// SIMATIC STEP 7 (V5.x) project Estacion completa
// CPU: CPU 314IFM
// station: P_ADR_BUS
// station: Hardware
// station: Equipo SIMATIC 300
// program: Programa S7(2)

// (several symbol tables fit these blocks; global names not applied)

DATA_BLOCK DB 1
VERSION : 0.1
  STRUCT
   M10 : BOOL ;	//Variable comodín provisional
  END_STRUCT ;	
BEGIN
END_DATA_BLOCK

ORGANIZATION_BLOCK OB 1
TITLE = "Main Program Sweep (Cycle)"
VERSION : 0.1
VAR_TEMP
  OB1_EV_CLASS : BYTE ;	//Bits 0-3 = 1 (Coming event), Bits 4-7 = 1 (Event class 1)
  OB1_SCAN_1 : BYTE ;	//1 (Cold restart scan 1 of OB 1), 3 (Scan 2-n of OB 1)
  OB1_PRIORITY : BYTE ;	//Priority of OB Execution
  OB1_OB_NUMBR : BYTE ;	//1 (Organization block 1, OB1)
  OB1_RESERVED_1 : BYTE ;	//Reserved for system
  OB1_RESERVED_2 : BYTE ;	//Reserved for system
  OB1_PREV_CYCLE : INT ;	//Cycle time of previous OB1 scan (milliseconds)
  OB1_MIN_CYCLE : INT ;	//Minimum cycle time of OB1 (milliseconds)
  OB1_MAX_CYCLE : INT ;	//Maximum cycle time of OB1 (milliseconds)
  OB1_DATE_TIME : DATE_AND_TIME ;	//Date and time OB1 started
END_VAR
BEGIN
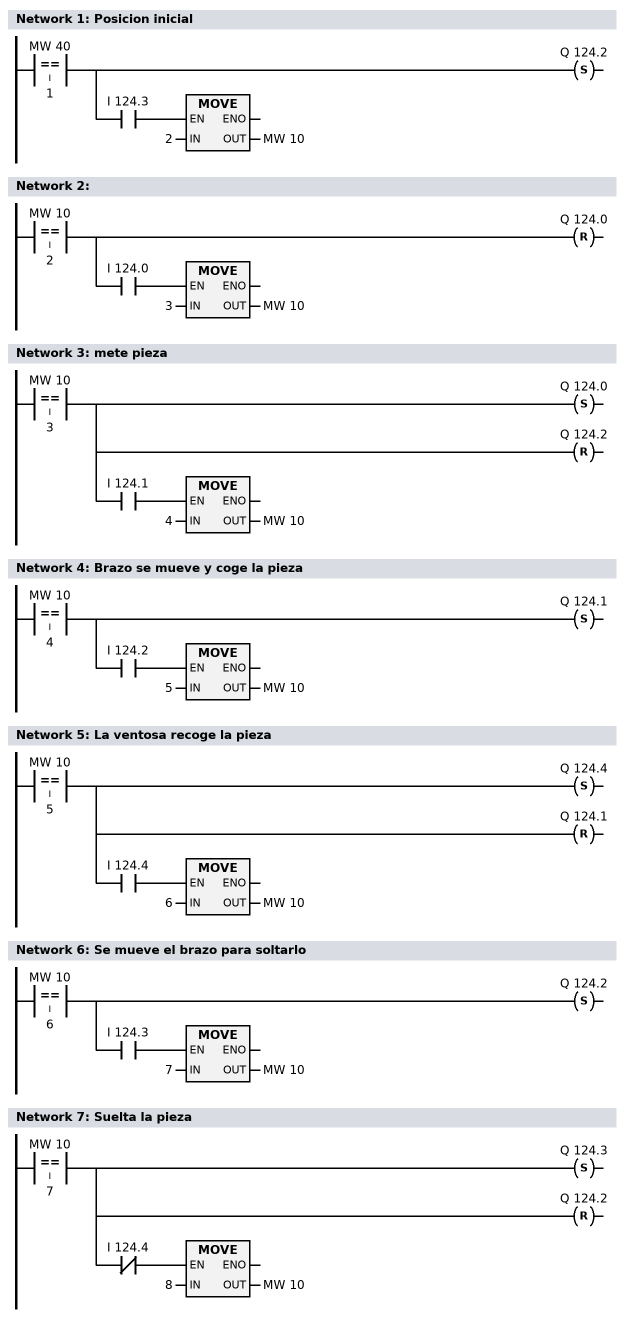
NETWORK
TITLE = Posicion inicial
      L     MW 40;
      L     1;
      ==I;
      =     L 20.0;
      A     L 20.0;
      BLD   102;
      S     Q 124.2;
      A     L 20.0;
      A     I 124.3;
      JNB   _001;
      L     2;
      T     MW 10;
_001: NOP   0;
NETWORK
TITLE =
      L     MW 10;
      L     2;
      ==I;
      =     L 20.0;
      A     L 20.0;
      BLD   102;
      R     Q 124.0;
      A     L 20.0;
      A     I 124.0;
      JNB   _002;
      L     3;
      T     MW 10;
_002: NOP   0;
NETWORK
TITLE = mete pieza
      L     MW 10;
      L     3;
      ==I;
      =     L 20.0;
      A     L 20.0;
      BLD   102;
      S     Q 124.0;
      A     L 20.0;
      BLD   102;
      R     Q 124.2;
      A     L 20.0;
      A     I 124.1;
      JNB   _003;
      L     4;
      T     MW 10;
_003: NOP   0;
NETWORK
TITLE = Brazo se mueve y coge la pieza
      L     MW 10;
      L     4;
      ==I;
      =     L 20.0;
      A     L 20.0;
      BLD   102;
      S     Q 124.1;
      A     L 20.0;
      A     I 124.2;
      JNB   _004;
      L     5;
      T     MW 10;
_004: NOP   0;
NETWORK
TITLE = La ventosa recoge la pieza
      L     MW 10;
      L     5;
      ==I;
      =     L 20.0;
      A     L 20.0;
      BLD   102;
      S     Q 124.4;
      A     L 20.0;
      BLD   102;
      R     Q 124.1;
      A     L 20.0;
      A     I 124.4;
      JNB   _005;
      L     6;
      T     MW 10;
_005: NOP   0;
NETWORK
TITLE = Se mueve el brazo para soltarlo
      L     MW 10;
      L     6;
      ==I;
      =     L 20.0;
      A     L 20.0;
      BLD   102;
      S     Q 124.2;
      A     L 20.0;
      A     I 124.3;
      JNB   _006;
      L     7;
      T     MW 10;
_006: NOP   0;
NETWORK
TITLE = Suelta la pieza
      L     MW 10;
      L     7;
      ==I;
      =     L 20.0;
      A     L 20.0;
      BLD   102;
      S     Q 124.3;
      A     L 20.0;
      BLD   102;
      R     Q 124.2;
      A     L 20.0;
      AN    I 124.4;
      JNB   _007;
      L     8;
      T     MW 10;
_007: NOP   0;
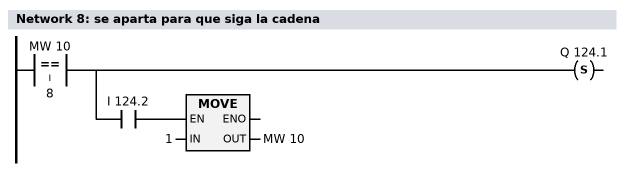
NETWORK
TITLE = se aparta para que siga la cadena
      L     MW 10;
      L     8;
      ==I;
      =     L 20.0;
      A     L 20.0;
      BLD   102;
      S     Q 124.1;
      A     L 20.0;
      A     I 124.2;
      JNB   _008;
      L     1;
      T     MW 10;
_008: NOP   0;
NETWORK
TITLE =
NETWORK
TITLE =
NETWORK
TITLE =
NETWORK
TITLE =
END_ORGANIZATION_BLOCK

SYMBOL_TABLE
"ATT"	FC 84	FC 84	// Add to Table
"CYCL_EXC"	OB 1	OB 1	// Cycle Execution
"COMPLETE RESTART"	OB 100	OB 100	// Complete Restart
"VAT_1"	VAT 1	
END_SYMBOL_TABLE

FUNCTION_BLOCK FB 1
VERSION : 0.1
BEGIN
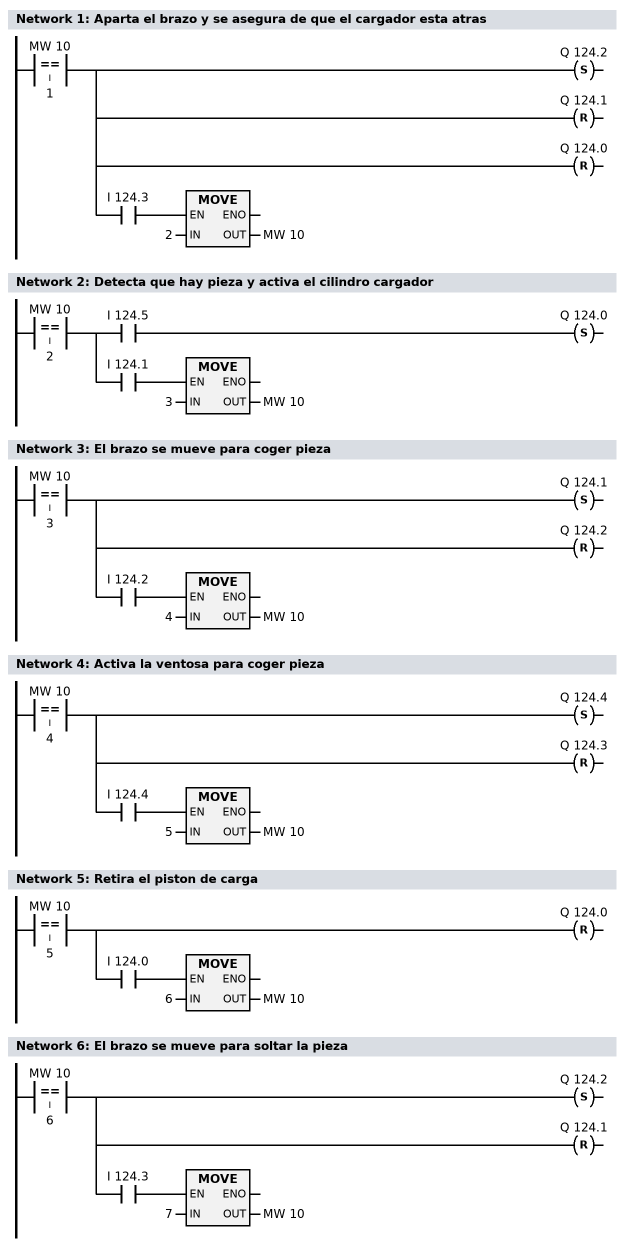
NETWORK
TITLE = Aparta el brazo y se asegura de que el cargador esta atras
      L     MW 10;
      L     1;
      ==I;
      =     L 0.0;
      A     L 0.0;
      BLD   102;
      S     Q 124.2;
      A     L 0.0;
      BLD   102;
      R     Q 124.1;
      A     L 0.0;
      BLD   102;
      R     Q 124.0;
      A     L 0.0;
      A     I 124.3;
      JNB   _001;
      L     2;
      T     MW 10;
_001: NOP   0;
NETWORK
TITLE = Detecta que hay pieza y activa el cilindro cargador
      L     MW 10;
      L     2;
      ==I;
      =     L 0.0;
      A     L 0.0;
      A     I 124.5;
      S     Q 124.0;
      A     L 0.0;
      A     I 124.1;
      JNB   _002;
      L     3;
      T     MW 10;
_002: NOP   0;
NETWORK
TITLE = El brazo se mueve para coger pieza
      L     MW 10;
      L     3;
      ==I;
      =     L 0.0;
      A     L 0.0;
      BLD   102;
      S     Q 124.1;
      A     L 0.0;
      BLD   102;
      R     Q 124.2;
      A     L 0.0;
      A     I 124.2;
      JNB   _003;
      L     4;
      T     MW 10;
_003: NOP   0;
NETWORK
TITLE = Activa la ventosa para coger pieza
      L     MW 10;
      L     4;
      ==I;
      =     L 0.0;
      A     L 0.0;
      BLD   102;
      S     Q 124.4;
      A     L 0.0;
      BLD   102;
      R     Q 124.3;
      A     L 0.0;
      A     I 124.4;
      JNB   _004;
      L     5;
      T     MW 10;
_004: NOP   0;
NETWORK
TITLE = Retira el piston de carga
      L     MW 10;
      L     5;
      ==I;
      =     L 0.0;
      A     L 0.0;
      BLD   102;
      R     Q 124.0;
      A     L 0.0;
      A     I 124.0;
      JNB   _005;
      L     6;
      T     MW 10;
_005: NOP   0;
NETWORK
TITLE = El brazo se mueve para soltar la pieza
      L     MW 10;
      L     6;
      ==I;
      =     L 0.0;
      A     L 0.0;
      BLD   102;
      S     Q 124.2;
      A     L 0.0;
      BLD   102;
      R     Q 124.1;
      A     L 0.0;
      A     I 124.3;
      JNB   _006;
      L     7;
      T     MW 10;
_006: NOP   0;
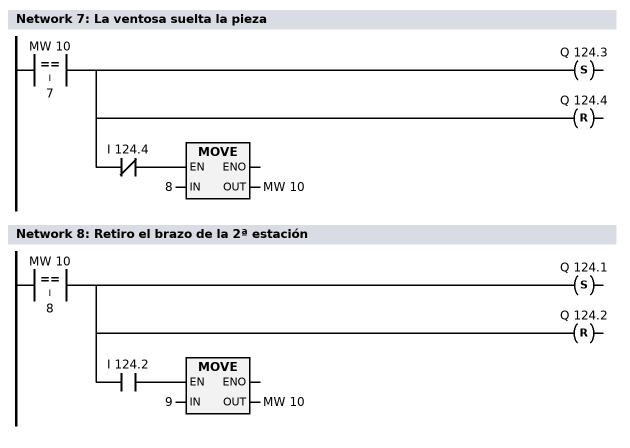
NETWORK
TITLE = La ventosa suelta la pieza
      L     MW 10;
      L     7;
      ==I;
      =     L 0.0;
      A     L 0.0;
      BLD   102;
      S     Q 124.3;
      A     L 0.0;
      BLD   102;
      R     Q 124.4;
      A     L 0.0;
      AN    I 124.4;
      JNB   _007;
      L     8;
      T     MW 10;
_007: NOP   0;
NETWORK
TITLE = Retiro el brazo de la 2ª estación
      L     MW 10;
      L     8;
      ==I;
      =     L 0.0;
      A     L 0.0;
      BLD   102;
      S     Q 124.1;
      A     L 0.0;
      BLD   102;
      R     Q 124.2;
      A     L 0.0;
      A     I 124.2;
      JNB   _008;
      L     9;
      T     MW 10;
_008: NOP   0;
END_FUNCTION_BLOCK

// FC 84: know-how protected block, not included

DATA_BLOCK DB 1
VERSION : 0.1
  STRUCT
   RP : INT ;	//Rojas pedidas
   RT : INT ;	//Rojas totales
   NP : INT ;	//Negras pedidas
   NT : INT ;	//Negras totales
   MP : INT ;	//Metalicas pedidas
   MT : INT ;	//Metalicas totales
   TBL : INT  := 10;	//Tabla de orden
   Cont : INT ;	//Contador de la tabla
   V1 : INT ;
   V2 : INT ;
   V3 : INT ;
   V4 : INT ;
   V5 : INT ;
   V6 : INT ;
   V7 : INT ;
   V8 : INT ;
   V9 : INT ;
  END_STRUCT ;	
BEGIN
   TBL := 10;
END_DATA_BLOCK

DATA_BLOCK DB 2
VERSION : 0.0
FB 1
BEGIN
END_DATA_BLOCK

ORGANIZATION_BLOCK "CYCL_EXC"	// OB 1
TITLE = "Main Program Sweep (Cycle)"
VERSION : 0.1
VAR_TEMP
  OB1_EV_CLASS : BYTE ;	//Bits 0-3 = 1 (Coming event), Bits 4-7 = 1 (Event class 1)
  OB1_SCAN_1 : BYTE ;	//1 (Cold restart scan 1 of OB 1), 3 (Scan 2-n of OB 1)
  OB1_PRIORITY : BYTE ;	//Priority of OB Execution
  OB1_OB_NUMBR : BYTE ;	//1 (Organization block 1, OB1)
  OB1_RESERVED_1 : BYTE ;	//Reserved for system
  OB1_RESERVED_2 : BYTE ;	//Reserved for system
  OB1_PREV_CYCLE : INT ;	//Cycle time of previous OB1 scan (milliseconds)
  OB1_MIN_CYCLE : INT ;	//Minimum cycle time of OB1 (milliseconds)
  OB1_MAX_CYCLE : INT ;	//Maximum cycle time of OB1 (milliseconds)
  OB1_DATE_TIME : DATE_AND_TIME ;	//Date and time OB1 started
END_VAR
BEGIN
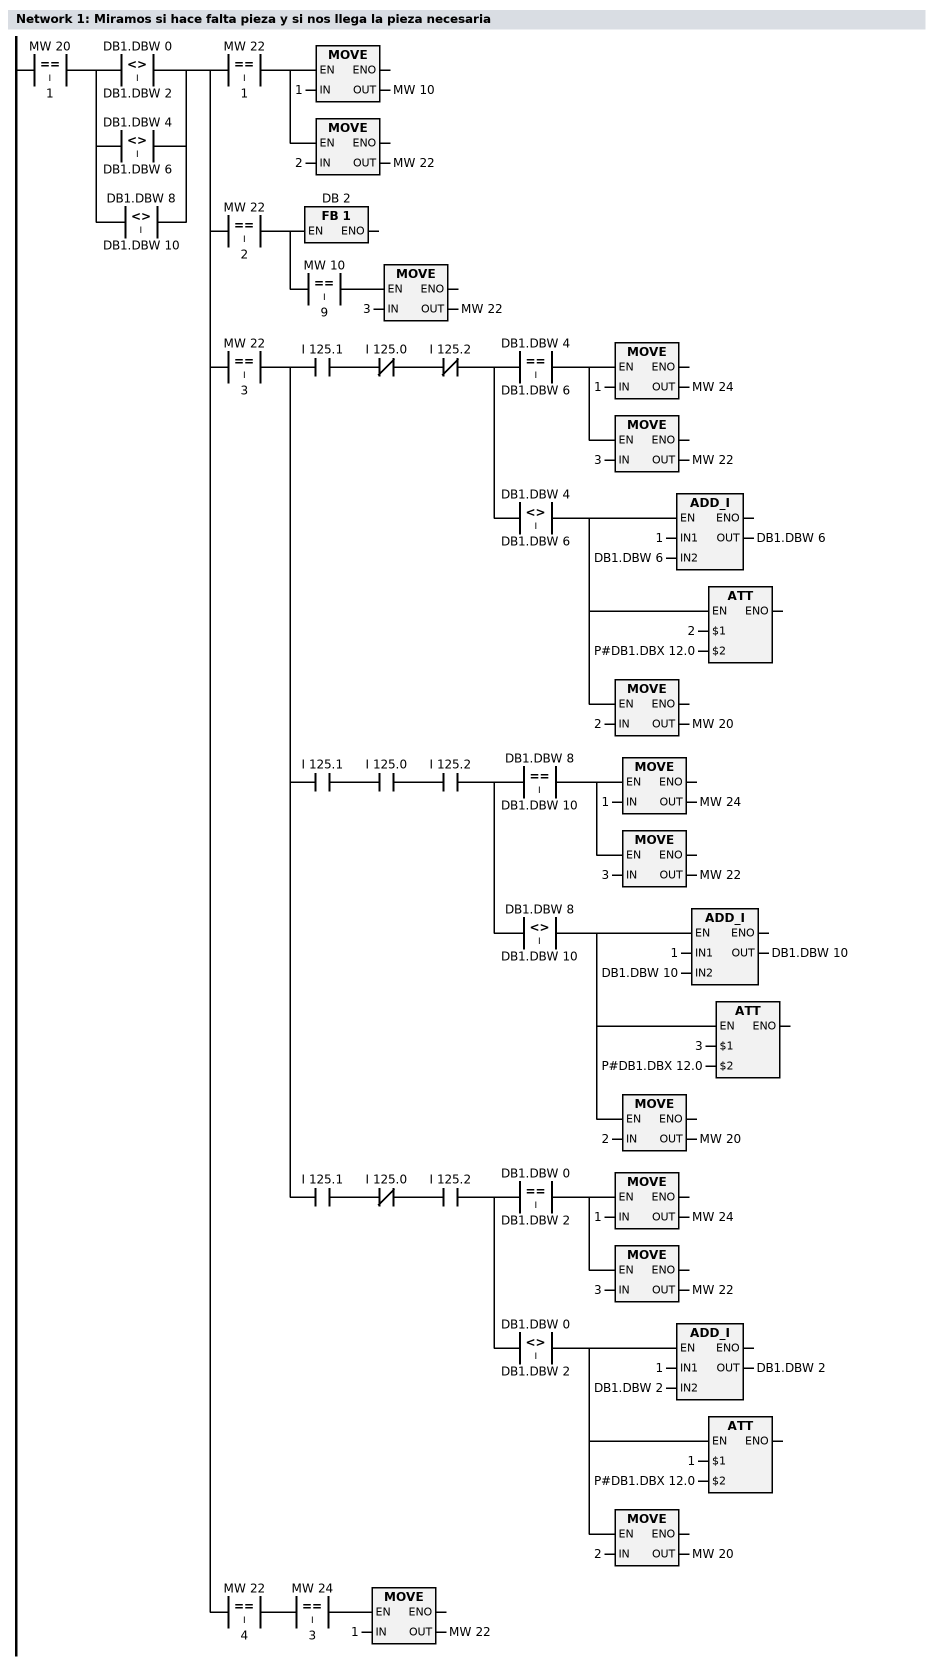
NETWORK
TITLE = Miramos si hace falta pieza y si nos llega la pieza necesaria
      A(;
      L     MW 20;
      L     1;
      ==I;
      );
      A(;
      O(;
      L     DB1.DBW 0;
      L     DB1.DBW 2;
      <>I;
      );
      O(;
      L     DB1.DBW 4;
      L     DB1.DBW 6;
      <>I;
      );
      O(;
      L     DB1.DBW 8;
      L     DB1.DBW 10;
      <>I;
      );
      );
      =     L 20.0;
      A     L 20.0;
      A(;
      L     MW 22;
      L     1;
      ==I;
      );
      =     L 20.1;
      A     L 20.1;
      JNB   _001;
      L     1;
      T     MW 10;
_001: NOP   0;
      A     L 20.1;
      JNB   _002;
      L     2;
      T     MW 22;
_002: NOP   0;
      A     L 20.0;
      A(;
      L     MW 22;
      L     2;
      ==I;
      );
      =     L 20.1;
      A     L 20.1;
      JNB   _003;
      CALL  FB 1 , DB 2;
_003: NOP   0;
      A     L 20.1;
      A(;
      L     MW 10;
      L     9;
      ==I;
      );
      JNB   _004;
      L     3;
      T     MW 22;
_004: NOP   0;
      A     L 20.0;
      A(;
      L     MW 22;
      L     3;
      ==I;
      );
      =     L 20.1;
      A     L 20.1;
      A     I 125.1;
      AN    I 125.0;
      AN    I 125.2;
      =     L 20.2;
      A     L 20.2;
      A(;
      L     DB1.DBW 4;
      L     DB1.DBW 6;
      ==I;
      );
      =     L 20.3;
      A     L 20.3;
      JNB   _005;
      L     1;
      T     MW 24;
_005: NOP   0;
      A     L 20.3;
      JNB   _006;
      L     3;
      T     MW 22;
_006: NOP   0;
      A     L 20.2;
      A(;
      L     DB1.DBW 4;
      L     DB1.DBW 6;
      <>I;
      );
      =     L 20.3;
      A     L 20.3;
      JNB   _007;
      L     1;
      L     DB1.DBW 6;
      +I;
      T     DB1.DBW 6;
_007: NOP   0;
      A     L 20.3;
      JNB   _008;
      CALL  "ATT" (
           $1                       := 2,
           $2                       := P#DB1.DBX 12.0);
_008: NOP   0;
      A     L 20.3;
      JNB   _009;
      L     2;
      T     MW 20;
_009: NOP   0;
      A     L 20.1;
      A     I 125.1;
      A     I 125.0;
      A     I 125.2;
      =     L 20.2;
      A     L 20.2;
      A(;
      L     DB1.DBW 8;
      L     DB1.DBW 10;
      ==I;
      );
      =     L 20.3;
      A     L 20.3;
      JNB   _00a;
      L     1;
      T     MW 24;
_00a: NOP   0;
      A     L 20.3;
      JNB   _00b;
      L     3;
      T     MW 22;
_00b: NOP   0;
      A     L 20.2;
      A(;
      L     DB1.DBW 8;
      L     DB1.DBW 10;
      <>I;
      );
      =     L 20.3;
      A     L 20.3;
      JNB   _00c;
      L     1;
      L     DB1.DBW 10;
      +I;
      T     DB1.DBW 10;
_00c: NOP   0;
      A     L 20.3;
      JNB   _00d;
      CALL  "ATT" (
           $1                       := 3,
           $2                       := P#DB1.DBX 12.0);
_00d: NOP   0;
      A     L 20.3;
      JNB   _00e;
      L     2;
      T     MW 20;
_00e: NOP   0;
      A     L 20.1;
      A     I 125.1;
      AN    I 125.0;
      A     I 125.2;
      =     L 20.2;
      A     L 20.2;
      A(;
      L     DB1.DBW 0;
      L     DB1.DBW 2;
      ==I;
      );
      =     L 20.3;
      A     L 20.3;
      JNB   _00f;
      L     1;
      T     MW 24;
_00f: NOP   0;
      A     L 20.3;
      JNB   _010;
      L     3;
      T     MW 22;
_010: NOP   0;
      A     L 20.2;
      A(;
      L     DB1.DBW 0;
      L     DB1.DBW 2;
      <>I;
      );
      =     L 20.3;
      A     L 20.3;
      JNB   _011;
      L     1;
      L     DB1.DBW 2;
      +I;
      T     DB1.DBW 2;
_011: NOP   0;
      A     L 20.3;
      JNB   _012;
      CALL  "ATT" (
           $1                       := 1,
           $2                       := P#DB1.DBX 12.0);
_012: NOP   0;
      A     L 20.3;
      JNB   _013;
      L     2;
      T     MW 20;
_013: NOP   0;
      A     L 20.0;
      A(;
      L     MW 22;
      L     4;
      ==I;
      );
      A(;
      L     MW 24;
      L     3;
      ==I;
      );
      JNB   _014;
      L     1;
      T     MW 22;
_014: NOP   0;
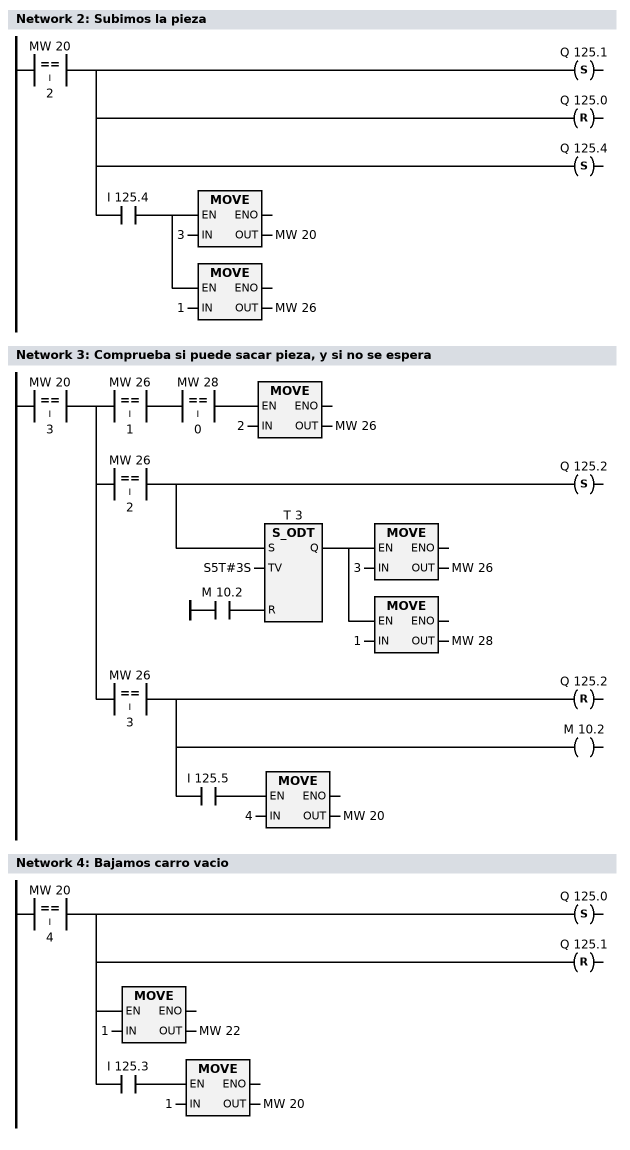
NETWORK
TITLE = Subimos la pieza
      L     MW 20;
      L     2;
      ==I;
      =     L 20.0;
      A     L 20.0;
      BLD   102;
      S     Q 125.1;
      A     L 20.0;
      BLD   102;
      R     Q 125.0;
      A     L 20.0;
      BLD   102;
      S     Q 125.4;
      A     L 20.0;
      A     I 125.4;
      =     L 20.1;
      A     L 20.1;
      JNB   _015;
      L     3;
      T     MW 20;
_015: NOP   0;
      A     L 20.1;
      JNB   _016;
      L     1;
      T     MW 26;
_016: NOP   0;
NETWORK
TITLE = Comprueba si puede sacar pieza, y si no se espera
      L     MW 20;
      L     3;
      ==I;
      =     L 20.0;
      A     L 20.0;
      A(;
      L     MW 26;
      L     1;
      ==I;
      );
      A(;
      L     MW 28;
      L     0;
      ==I;
      );
      JNB   _017;
      L     2;
      T     MW 26;
_017: NOP   0;
      A     L 20.0;
      A(;
      L     MW 26;
      L     2;
      ==I;
      );
      =     L 20.1;
      A     L 20.1;
      BLD   102;
      S     Q 125.2;
      A     L 20.1;
      L     S5T#3S;
      SD    T 3;
      A     M 10.2;
      R     T 3;
      NOP   0;
      NOP   0;
      A     T 3;
      =     L 20.2;
      A     L 20.2;
      JNB   _018;
      L     3;
      T     MW 26;
_018: NOP   0;
      A     L 20.2;
      JNB   _019;
      L     1;
      T     MW 28;
_019: NOP   0;
      A     L 20.0;
      A(;
      L     MW 26;
      L     3;
      ==I;
      );
      =     L 20.1;
      A     L 20.1;
      BLD   102;
      R     Q 125.2;
      A     L 20.1;
      BLD   102;
      =     M 10.2;
      A     L 20.1;
      A     I 125.5;
      JNB   _01a;
      L     4;
      T     MW 20;
_01a: NOP   0;
NETWORK
TITLE = Bajamos carro vacio
      L     MW 20;
      L     4;
      ==I;
      =     L 20.0;
      A     L 20.0;
      BLD   102;
      S     Q 125.0;
      A     L 20.0;
      BLD   102;
      R     Q 125.1;
      A     L 20.0;
      JNB   _01b;
      L     1;
      T     MW 22;
_01b: NOP   0;
      A     L 20.0;
      A     I 125.3;
      JNB   _01c;
      L     1;
      T     MW 20;
_01c: NOP   0;
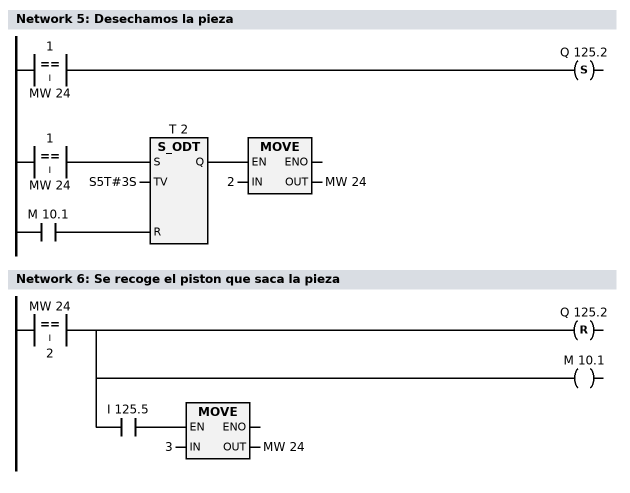
NETWORK
TITLE = Desechamos la pieza
      L     1;
      L     MW 24;
      ==I;
      =     L 20.0;
      A     L 20.0;
      BLD   102;
      S     Q 125.2;
      A(;
      A     L 20.0;
      L     S5T#3S;
      SD    T 2;
      A     M 10.1;
      R     T 2;
      NOP   0;
      NOP   0;
      A     T 2;
      );
      JNB   _01d;
      L     2;
      T     MW 24;
_01d: NOP   0;
NETWORK
TITLE = Se recoge el piston que saca la pieza
      L     MW 24;
      L     2;
      ==I;
      =     L 20.0;
      A     L 20.0;
      BLD   102;
      R     Q 125.2;
      A     L 20.0;
      BLD   102;
      =     M 10.1;
      A     L 20.0;
      A     I 125.5;
      JNB   _01e;
      L     3;
      T     MW 24;
_01e: NOP   0;
END_ORGANIZATION_BLOCK

SYMBOL_TABLE
"Cycle Execution"	OB 1	OB 1
"COMPLETE RESTART"	OB 100	OB 100	// Complete Restart
"VAT_1"	VAT 1	
END_SYMBOL_TABLE
